# EPICS autosave request: iocBoot/sioc-li21-im02/adc_manual.req
file "manual.req" AREA=LI21,POS=206
file "manual.req" AREA=LI21,POS=278
